// TIA Portal project "HMI_PROJECT" (V16)

(* hardware
DEVICE "S7300/ET200M station_1"  S7-300 station
   slot 0: "Rail_0"  Rail  6ES7 390-1***0-0AA0
   slot 2: "PLC_1"  CPU 314C-2 DP  6ES7 314-6CH04-0AB0  V3.3
      slot 0: "MPI interface_1"  MPI
      slot 1: "DP interface_1"  DP
      slot 2: "DI 24/DO 16_1"  DI24/DO16
      slot 3: "AI 5/AO 2_1"  AI5/AO2
      slot 4: "Count_1"  Counter
      slot 5: "Positioning_1"  Positioning
   slot 4: "DI 16x24VDC_1"  DI16 x 24VDC  6ES7 321-1BH50-0AA0
   slot 5: "DO 8x24VDC/0.5A_1"  DO8 x 24VDC / 0.5A  6ES7 322-8BF00-0AB0
DEVICE "HMI_1"  KTP700 Basic DP
   slot 0: "HMI_1"  KTP700 Basic DP  6AV2 123-2GA03-0AX0  16.0.0.0
   slot 1: "HMI_RT_1"  KTP700 Basic DP  6AV2 123-2GA03-0AX0  16.0.0.0
   slot 7: "HMI_1.MPI/DP_CP_1"  MPI/DP Interface  16.0.0.0
*)

// ===== PLC "PLC_1"  CPU 314C-2 DP =====

VAR_GLOBAL   // PLC tag table "Default tag table"
   "START1" AT %M0.0 : Bool;
   "STOPGENERAL" AT %M0.1 : Bool;
   "MOTOR1" AT %Q0.0 : Bool;
   "MOTOR2" AT %Q0.1 : Bool;
   "START2" AT %M0.2 : Bool;
END_VAR

ORGANIZATION_BLOCK "Main"   // OB1, LAD
TITLE = "Main Program Sweep (Cycle)"
{ S7_Optimized_Access := 'FALSE' }
VERSION : 0.1
   VAR_TEMP
      OB1_EV_CLASS : Byte;   // Bits 0-3 = 1 (Coming event), Bits 4-7 = 1 (Event class 1)
      OB1_SCAN_1 : Byte;   // 1 (Cold restart scan 1 of OB 1), 3 (Scan 2-n of OB 1)
      OB1_PRIORITY : Byte;   // Priority of OB Execution
      OB1_OB_NUMBR : Byte;   // 1 (Organization block 1, OB1)
      OB1_RESERVED_1 : Byte;   // Reserved for system
      OB1_RESERVED_2 : Byte;   // Reserved for system
      OB1_PREV_CYCLE : Int;   // Cycle time of previous OB1 scan (milliseconds)
      OB1_MIN_CYCLE : Int;   // Minimum cycle time of OB1 (milliseconds)
      OB1_MAX_CYCLE : Int;   // Maximum cycle time of OB1 (milliseconds)
      OB1_DATE_TIME : Date_And_Time;   // Date and time OB1 started
   END_VAR
BEGIN

REGION Network 1
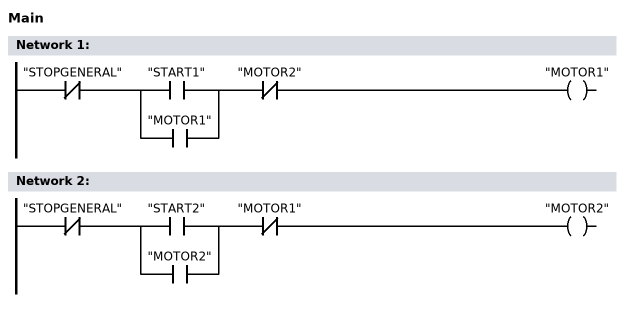
   RUNG wire#powerrail
      I_Contact( "STOPGENERAL" )
      wire#w1
      Contact( "START1" )
      wire#w2
      I_Contact( "MOTOR2" )
      Coil( "MOTOR1" )
   END_RUNG
   RUNG wire#w1
      Contact( "MOTOR1" )
   END_RUNG wire#w2
   // the same network as SCL:
   "MOTOR1" := NOT "STOPGENERAL" AND ("START1" OR "MOTOR1") AND NOT "MOTOR2";
END_REGION

REGION Network 2
   RUNG wire#powerrail
      I_Contact( "STOPGENERAL" )
      wire#w1
      Contact( "START2" )
      wire#w2
      I_Contact( "MOTOR1" )
      Coil( "MOTOR2" )
   END_RUNG
   RUNG wire#w1
      Contact( "MOTOR2" )
   END_RUNG wire#w2
   // the same network as SCL:
   "MOTOR2" := NOT "STOPGENERAL" AND ("START2" OR "MOTOR2") AND NOT "MOTOR1";
END_REGION
END_ORGANIZATION_BLOCK

(* ===== HMI "HMI_RT_1" =====
system functions are stored by id; their names below are inferred from use
connection "HMI_Connection_1": IF1 B, SIMATIC S7 300/400 MPI
connection "HMI_Connection_2": IF1 B, SIMATIC S7 300/400 MPI

HMI tags "Default tag table"
   "ARRANQUE1" : Bool = PLC START1 AT %M0.0, 1 s
   "ARRANQUE2" : Bool = PLC START2 AT %M0.2, 1 s
   "PAROGENERAL" : Bool = PLC STOPGENERAL AT %M0.1, 1 s
   "MOTOR1" : Bool = PLC MOTOR1 AT %Q0.0, 1 s
   "MOTOR2" : Bool = PLC MOTOR2 AT %Q0.1, 1 s
   "START_1_1" : Bool = PLC START1 AT %M0.0, 1 s
   "START_1_2" : Bool = PLC START2 AT %M0.2, 1 s
   "STOPGENERAL" : Bool = PLC STOPGENERAL AT %M0.1, 1 s

screen "Root screen_1" 800x480
   GraphicView "Graphic view_1" at 0,0 size 800x60; Picture "Página inicial HMI"
   TextField "Text field_1" at 641,164 size 101x32; Text 'MOTOR 1'
   TextField "Text field_2" at 641,257 size 101x32; Text 'MOTOR 2'
   TextField "Text field_3" at 664,341 size 59x32; Text 'STOP'
   TextField "Text field_4" at 515,99 size 249x32; Text 'CONTROL DE MOTORES'
   GraphicView "Graphic view_2" at 23,137 size 128x128; Picture "electric-motor _OFF"
      Visibility <- "MOTOR1"
   GraphicView "Graphic view_3" at 23,137 size 128x128; Picture "electric-motor_ON"
      Visibility <- "MOTOR1"
   GraphicView "Graphic view_4" at 27,263 size 128x128; Picture "electric-motor _OFF"
      Visibility <- "MOTOR2"
   GraphicView "Graphic view_5" at 27,263 size 128x128; Picture "electric-motor_ON"
      Visibility <- "MOTOR2"
   TextField "Text field_5" at 190,192 size 101x32; Text 'MOTOR 1'
   TextField "Text field_6" at 194,304 size 101x32; Text 'MOTOR 2'
   TextField "Text field_7" at 144,80 size 114x32; Text 'MOTORES'
   Button "Button_1" at 511,175 size 96x32; TextOff 'MOTOR 1'
      on Press: function_b14e0dd5("ARRANQUE1", 0)
   Button "Button_2" at 511,260 size 96x32; TextOff 'MOTOR 2'
      on Press: function_b14e0dd5("ARRANQUE2", 0)
   Button "Button_3" at 515,342 size 96x32; TextOff 'PARADA'
      on Press: function_b14e0dd5("PAROGENERAL", 0)
*)